// TwinCAT 3 PLC project SEFrey_StringBuilder
// Title: StringBuilder
// Company: S.E.Frey
// Author: Michi
// ProjectVersion: 0.01
// Description: Simple but powerfull stringbuilder, working with any in TC3 available datatype
// ProgramVersion: 3.1.4024.0
// libraries:
//   Tc2_Standard, * (Beckhoff Automation GmbH)
//   Tc2_System, * (Beckhoff Automation GmbH)
//   Tc2_Utilities, * (Beckhoff Automation GmbH)
//   Tc3_Module, * (Beckhoff Automation GmbH)
// project tree:
//   DUTs/ ST_StringBuilderPara.TcDUT
//   GVLs/ GVL_StringBuilder.TcGVL
//   / PlcTask.TcTTO
//   POUs/ MAIN.TcPOU
//   POUs/StringBuilder/ CStringBuilder.TcPOU
//   POUs/StringBuilder/Examples/ CStringBuilderExample.TcPOU
//   POUs/StringBuilder/Functions/ BuildString.TcPOU
//   POUs/StringBuilder/Interfaces/ I_StringBuilder.TcIO
// real-time tasks:
//   TASK PlcTask: cycle T#10ms, priority 20, ADS port 350

CONFIGURATION SEFrey_StringBuilder
    RESOURCE PLC ON TwinCAT3
        TASK PlcTask(INTERVAL := T#10ms, PRIORITY := 20);
        PROGRAM MAIN WITH PlcTask : MAIN;
    END_RESOURCE
END_CONFIGURATION

// ---- DUTs/ST_StringBuilderPara.TcDUT
{attribute 'enable_dynamic_creation'}
TYPE ST_StringBuilderPara :
STRUCT
	MaxBufferSize : UDINT; //defines max possible string length
END_STRUCT
END_TYPE

// ---- GVLs/GVL_StringBuilder.TcGVL
{attribute 'qualified_only'}
VAR_GLOBAL
	pStringBuilder : POINTER TO CStringBuilder;
	pPara : POINTER TO ST_StringBuilderPara;
END_VAR

// ---- POUs/StringBuilder/Interfaces/I_StringBuilder.TcIO
INTERFACE I_StringBuilder

METHOD Append : I_StringBuilder
VAR_INPUT
	Value : T_MaxString;
END_VAR
END_METHOD

METHOD AppendAny : I_StringBuilder
VAR_INPUT
	Value : ANY;
END_VAR
END_METHOD

PROPERTY BufferAddress : POINTER TO BYTE
GET
END_GET
END_PROPERTY

METHOD Clear : I_StringBuilder
VAR_INPUT
END_VAR
END_METHOD

END_INTERFACE

// ---- POUs/MAIN.TcPOU
PROGRAM MAIN
VAR
	StringBuilderExample : CStringBuilderExample;
END_VAR

StringBuilderExample.ClassAndInitialization();
StringBuilderExample.SimpleUse();

END_PROGRAM

// ---- POUs/StringBuilder/Examples/CStringBuilderExample.TcPOU
FUNCTION_BLOCK CStringBuilderExample
VAR_INPUT
END_VAR
VAR_OUTPUT
END_VAR
VAR
	//run tests
	startClassAndInitializationTest, startSimpleUseTest : BOOL;

	
	simpleUseOutput1, simpleUseOutput2 : STRING(200);

	
	StringBuilder : CStringBuilder; //500 characters + 0 terminator (/0)
	Value : STRING(255) := 'Dieser Text ist genau 250 Zeichen lang und wird verwendet, um zu zeigen, wie TwinCAT 3 Strings handhabt. Es handelt sich um einen langen Satz, der viele verschiedene Themen behandelt, wie z.B. Programmierung, Automatisierungstechnik, SPS-Programmieru';
	currentString:  STRING(3000);
	pResult : POINTER TO BYTE;
	Stage, SimpleUseStage : INT;
	
	stStringBuilderPara : ST_StringBuilderPara := (MaxBufferSize:=3000);
	
 	boolExample : BOOL := TRUE;
    byteExample : BYTE := 16#FF;
    wordExample : WORD := 16#FFFF;
    dwordExample : DWORD := 16#FFFFFFFF;
    lwordExample : LWORD := 16#FFFFFFFFFFFFFFFF;
    sintExample : SINT := -128;
    intExample : INT := -32768;
    dintExample : DINT := -2147483648;
    lintExample : LINT := -9223372036854775808;
    usintExample : USINT := 255;
    uintExample : UINT := 65535;
    udintExample : UDINT := 4294967295;
    ulintExample : ULINT := 18446744073709551615;
    realExample : REAL := 1.0;
    lrealExample : LREAL := 1.0;
    timeExample : TIME := T#5s;
    dateExample : DATE := D#2023-01-01;
    todExample : TOD := TOD#12:00:00;
    dtExample : DT := DT#2023-01-01-12:00:00;
    stringExample : STRING := 'I am a string';
END_VAR

METHOD ClassAndInitialization : BOOL
VAR_INPUT
END_VAR
CASE Stage OF
	
	0:
		IF startClassAndInitializationTest THEN
			startClassAndInitializationTest := FALSE;
			StringBUilder.Init(pPara:=ADR(THIS^.stStringBuilderPara));
			Stage := 1;
		END_IF
		
	1:
		StringBuilder
            .Append(Value:='This is a bool: ')
            .AppendAny(Value:=boolExample)
            .Append(Value:=', This is a byte: ')
            .AppendAny(Value:=byteExample)
            .Append(Value:=', This is a word: ')
            .AppendAny(Value:=wordExample)
            .Append(Value:=', This is a dword: ')
            .AppendAny(Value:=dwordExample)
            .Append(Value:=', This is a lword: ')
            .AppendAny(Value:=lwordExample)
            .Append(Value:=', This is a sint: ')
            .AppendAny(Value:=sintExample)
            .Append(Value:=', This is an int: ')
            .AppendAny(Value:=intExample);
			
			//separation done, compiling + logging in needs pretty long for chains longer than 14
			StringBuilder
			.Append(Value:=', This is a dint: ')
            .AppendAny(Value:=dintExample)
            .Append(Value:=', This is a lint: ')
            .AppendAny(Value:=lintExample)
            .Append(Value:=', This is a usint: ')
            .AppendAny(Value:=usintExample)
            .Append(Value:=', This is a uint: ')
            .AppendAny(Value:=uintExample)
            .Append(Value:=', This is a udint: ')
            .AppendAny(Value:=udintExample)
            .Append(Value:=', This is a ulint: ')
            .AppendAny(Value:=ulintExample)
            .Append(Value:=', This is a real: ')
            .AppendAny(Value:=realExample);
			
			StringBuilder
            .Append(Value:=', This is an lreal: ')
            .AppendAny(Value:=lrealExample)
            .Append(Value:=', This is a time: ')
            .AppendAny(Value:=timeExample)
            .Append(Value:=', This is a date: ')
            .AppendAny(Value:=dateExample)
            .Append(Value:=', This is a tod: ')
            .AppendAny(Value:=todExample)
            .Append(Value:=', This is a dt: ')
            .AppendAny(Value:=dtExample)
            .Append(Value:=', This is a string: ')
            .AppendAny(Value:=stringExample);
		// show string data
		StringBuilder.Copy(pDest:=ADR(currentString), n:=SIZEOF(currentString));
		Stage := 2;
		
		2:
			StringBuilder.Clear();
			Stage := 0;
		
		
END_CASE
END_METHOD

METHOD SimpleUse : BOOL
VAR_INPUT
END_VAR
// build string, copy to destination

CASE SimpleUseStage OF


	0:
		IF THIS^.startSimpleUseTest THEN
			startSimpleUseTest := FALSE;
			//build string, copy to given destination
			BuildString(nSizeDest:=SIZEOF(simpleUseOutput1))
			.AppendAny(boolExample)
			.AppendAny(dintExample)
			.Copy(pDest:=ADR(simpleUseOutput1), n:=SIZEOF(simpleUseOutput1));
			SimpleUseStage := 1;
		END_IF
		
	1: //clear buffer, fill + copy to next string
		BuildString(nSizeDest:=SIZEOF(simpleUseOutput2))
		.Clear()
		.AppendAny(dwordExample)
		.AppendAny(dtExample)
		.AppendAny(stringExample)
		.Copy(pDest:=ADR(simpleUseOutput2), n:=SIZEOF(simpleUseOutput2));
		SimpleUseStage := 0;
	
	
	
	
END_CASE
END_METHOD

END_FUNCTION_BLOCK

// ---- POUs/StringBuilder/CStringBuilder.TcPOU
{attribute 'no_assign'}
{attribute 'enable_dynamic_creation'}
{attribute 'no_explicit_call' := 'do not call this POU directly'}
{attribute 'reflection'} 
FUNCTION_BLOCK CStringBuilder IMPLEMENTS I_StringBuilder
VAR_INPUT
END_VAR
VAR_OUTPUT
END_VAR
VAR
	pBuffer : POINTER TO BYTE;
	_maxBufferSize : UDINT; //defines max possible string length
	_currentUsedBufferSize : UDINT;
	
	{attribute 'instance-path'} 
    {attribute 'noinit'} 
    sPath : STRING; 
END_VAR

METHOD AnyToString : STRING
VAR_INPUT
	Value : ANY;
END_VAR
VAR
	pBool			: POINTER TO BOOL;
    pByte			: POINTER TO BYTE;
    pWord			: POINTER TO WORD;
    pDWord			: POINTER TO DWORD;
    pLWord			: POINTER TO LWORD;
    pSint			: POINTER TO SINT;
    pInt			: POINTER TO INT;
    pDint			: POINTER TO DINT;
    pLint			: POINTER TO LINT;
    pUSint			: POINTER TO USINT;
    pUInt			: POINTER TO UINT;
    pUDint			: POINTER TO UDINT;
    pULint			: POINTER TO ULINT;
    pReal			: POINTER TO REAL;
    pLReal			: POINTER TO LREAL;
    pString			: POINTER TO T_MaxString;
    pWString		: POINTER TO WSTRING;
    pTime			: POINTER TO TIME;
    pDate			: POINTER TO DATE;
    pDateAndTime	: POINTER TO DATE_AND_TIME;
    pTimeOfDay		: POINTER TO TIME_OF_DAY;
    pPointer		: PVOID;
	pLTime 			: POINTER TO LTIME;
END_VAR
IF Value.pValue = 0 THEN RETURN; END_IF;

CASE Value.TypeClass OF 
	__SYSTEM.TYPE_CLASS.TYPE_BOOL:
		pBool := Value.pValue;
		AnyToString := TO_STRING(pBool^);
		
    __SYSTEM.TYPE_CLASS.TYPE_BYTE:
		pByte := Value.pValue;
		AnyToString := TO_STRING(pByte^);
		
    __SYSTEM.TYPE_CLASS.TYPE_WORD:
		pWord := Value.pValue;
		AnyToString := TO_STRING(pWord^);
		
    __SYSTEM.TYPE_CLASS.TYPE_DWORD:
		pDWord := Value.pValue;
		AnyToString := TO_STRING(pDWord^);
		
    __SYSTEM.TYPE_CLASS.TYPE_LWORD:
		pLWord := Value.pValue;
		AnyToString := TO_STRING(pLWord^);
		
    __SYSTEM.TYPE_CLASS.TYPE_SINT:
		pSint := Value.pValue;
		AnyToString := TO_STRING(pSint^);
		
    __SYSTEM.TYPE_CLASS.TYPE_INT:
		pInt := Value.pValue;
		AnyToString := TO_STRING(pInt^);
		
    __SYSTEM.TYPE_CLASS.TYPE_DINT:
		pDint := Value.pValue;
		AnyToString := TO_STRING(pDint^);
		
    __SYSTEM.TYPE_CLASS.TYPE_LINT:
		pLint := Value.pValue;
		AnyToString := TO_STRING(pLint^);
		
    __SYSTEM.TYPE_CLASS.TYPE_USINT:
		pUSint := Value.pValue;
		AnyToString := TO_STRING(pUSint^);
		
    __SYSTEM.TYPE_CLASS.TYPE_UINT:
		pUInt := Value.pValue;
		AnyToString := TO_STRING(pUInt^);
		
    __SYSTEM.TYPE_CLASS.TYPE_UDINT:
		pUDint := Value.pValue;
		AnyToString := TO_STRING(pUDint^);
		
    __SYSTEM.TYPE_CLASS.TYPE_ULINT:
		pULint := Value.pValue;
		AnyToString := TO_STRING(pULint^);
		
   __SYSTEM.TYPE_CLASS.TYPE_REAL:
		pReal := Value.pValue;
		AnyToString := TO_STRING(pReal^);
		
    __SYSTEM.TYPE_CLASS.TYPE_LREAL:
		pLReal := Value.pValue;
		AnyToString := TO_STRING(pLReal^);
		
    __SYSTEM.TYPE_CLASS.TYPE_STRING:
		pString := Value.pValue;
		AnyToString := TO_STRING(pString^);
		
   __SYSTEM.TYPE_CLASS.TYPE_WSTRING:
		pWString := Value.pValue;
		AnyToString := TO_STRING(pWString^);
		
    __SYSTEM.TYPE_CLASS.TYPE_TIME:
		pTime := Value.pValue;
		AnyToString := TO_STRING(pTime^);
		
    __SYSTEM.TYPE_CLASS.TYPE_DATE:
		pDate := Value.pValue;
		AnyToString := TO_STRING(pDate^);
		
    __SYSTEM.TYPE_CLASS.TYPE_DATEANDTIME:
		pDateAndTime := Value.pValue;
		AnyToString := TO_STRING(pDateAndTime^);
		
    __SYSTEM.TYPE_CLASS.TYPE_TIMEOFDAY:
		pTimeOfDay := Value.pValue;
		AnyToString := TO_STRING(pTimeOfDay^);
	
	__SYSTEM.TYPE_CLASS.TYPE_POINTER:
		AnyToString := TO_STRING(Value.pValue);
		
	__SYSTEM.TYPE_CLASS.TYPE_LTIME:
		pLTime := Value.pValue;
		AnyToString := TO_STRING(pLTime^);
ELSE
	RETURN; 
END_CASE
END_METHOD

METHOD Append : I_StringBuilder
VAR_INPUT
	Value : T_MaxString;
END_VAR
Append := THIS^.AppendAny(Value);
END_METHOD

// Appends the given value to the end of the string builder's contents.
METHOD AppendAny : I_StringBuilder
VAR_INPUT
	Value : ANY;
END_VAR
VAR
	stringLength : UDINT;
	convertedAny : STRING; 
	pValue : POINTER TO BYTE;
END_VAR
AppendAny := THIS^;

IF THIS^.pBuffer = 0 THEN
	ADSLOGSTR(msgCtrlMask:= ADSLOG_MSGTYPE_ERROR, msgFmtStr:='Dynamic buffer null pointer, usage of StringBuilder not possible', '');
	RETURN;
END_IF

CASE Value.TypeClass OF
	__SYSTEM.TYPE_CLASS.TYPE_STRING: 
		pValue := Value.pValue;
		
	__SYSTEM.TYPE_CLASS.TYPE_BOOL,
	__SYSTEM.TYPE_CLASS.TYPE_BYTE,
	__SYSTEM.TYPE_CLASS.TYPE_WORD,
	__SYSTEM.TYPE_CLASS.TYPE_DWORD,
	__SYSTEM.TYPE_CLASS.TYPE_LWORD,
	__SYSTEM.TYPE_CLASS.TYPE_SINT,
	__SYSTEM.TYPE_CLASS.TYPE_INT,
	__SYSTEM.TYPE_CLASS.TYPE_DINT,
	__SYSTEM.TYPE_CLASS.TYPE_LINT,
	__SYSTEM.TYPE_CLASS.TYPE_USINT,
	__SYSTEM.TYPE_CLASS.TYPE_UINT,
	__SYSTEM.TYPE_CLASS.TYPE_UDINT,
	__SYSTEM.TYPE_CLASS.TYPE_ULINT,
	__SYSTEM.TYPE_CLASS.TYPE_REAL,
	__SYSTEM.TYPE_CLASS.TYPE_LREAL,
	__SYSTEM.TYPE_CLASS.TYPE_TIME,
	__SYSTEM.TYPE_CLASS.TYPE_LTIME,
	__SYSTEM.TYPE_CLASS.TYPE_DATE,
	__SYSTEM.TYPE_CLASS.TYPE_DATEANDTIME,
	__SYSTEM.TYPE_CLASS.TYPE_TIMEOFDAY,
	__SYSTEM.TYPE_CLASS.TYPE_POINTER:
		convertedAny := AnyToString(Value);
		pValue := ADR(convertedAny);
ELSE
	RETURN;
END_CASE

stringLength := GetUsedStringLength(pByte:=pValue);

//check available size, existing size
IF stringLength = 0 THEN
	RETURN;
END_IF
//only copy if we do not exceed possible limit
IF THIS^._currentUsedBufferSize + stringLength >= THIS^._maxBufferSize THEN
	RETURN;
END_IF
MEMCPY(destAddr:=(THIS^.pBuffer + THIS^._currentUsedBufferSize), srcAddr:=pValue, n:=stringLength);

THIS^._currentUsedBufferSize := THIS^._currentUsedBufferSize + stringLength;
END_METHOD

PROPERTY BufferAddress : POINTER TO BYTE
GET
BufferAddress := THIS^.pBuffer;
END_GET
END_PROPERTY

METHOD Clear : I_StringBuilder
VAR_INPUT
END_VAR
Clear := THIS^;
IF THIS^.pBuffer = 0 THEN
	RETURN;
END_IF

MEMSET(destAddr:=THIS^.pBuffer, fillByte:=0, n:=THIS^.MaxBufferSize);
_currentUsedBufferSize := 0;
END_METHOD

METHOD Copy : BOOL
VAR_INPUT
	pDest : POINTER TO BYTE;
	n : UDINT; // Size of destination
END_VAR
MEMCPY(destAddr:=pDest, srcAddr:=THIS^.BufferAddress, n:=n);
Copy := TRUE;
END_METHOD

PROPERTY CurrentBufferSize : UDINT
GET
CurrentBufferSize := THIS^._currentUsedBufferSize;
END_GET
END_PROPERTY

METHOD GetUsedStringLength : UDINT
VAR_INPUT
	pByte : POINTER TO BYTE;
END_VAR
VAR
    i : UDINT := 0;
END_VAR
//every string in twincat is 0 terminated
IF pByte = 0 THEN
	RETURN;
END_IF

WHILE (pByte^ <> 0) DO
    pByte := pByte + 1; // Pointer auf das nächste Byte verschieben
    i := i + 1;
END_WHILE;

GetUsedStringLength := i;
END_METHOD

METHOD Init : I_StringBuilder
VAR_INPUT
	pPara : POINTER TO ST_StringBuilderPara;
END_VAR
// TODO: add logging for failed allocation
IF ParaErrors(pPara:=pPara) THEN
	RETURN;
END_IF

IF THIS^.pBuffer <> 0 THEN
	__DELETE(THIS^.pBuffer);
END_IF

THIS^.pBuffer := __NEW(BYTE, pPara^.MaxBufferSize);
THIS^._maxBufferSize := pPara^.MaxBufferSize;
END_METHOD

PROPERTY MaxBufferSize : UDINT
GET
MaxBufferSize := THIS^._maxBufferSize;
END_GET
END_PROPERTY

{attribute 'reflection'} 
METHOD PRIVATE ParaErrors : BOOL
VAR_INPUT
	pPara : POINTER TO ST_StringBuilderPara;
END_VAR
VAR
	s1 : STRING(35) := 'Invalid parametrization pointer at ';
	s2: T_MaxString;
END_VAR
IF pPara = 0 THEN
	CONCAT2(pSrcString1:=ADR(s1), pSrcString2:=ADR(THIS^.sPath), pDstString:=ADR(s2), nDstSize:=SIZEOF(s2));
	ADSLOGSTR(msgCtrlMask:= ADSLOG_MSGTYPE_ERROR, msgFmtStr:=s2, '');
	ParaErrors := TRUE;
	RETURN;
END_IF
IF pPara^.MaxBufferSize = 0 THEN
	s1 := 'BufferSize 0 given, Stringbuilder init failed at ';
	CONCAT2(pSrcString1:=ADR(s1), pSrcString2:=ADR(THIS^.sPath), pDstString:=ADR(s2), nDstSize:=SIZEOF(s2));
	ADSLOGSTR(msgCtrlMask:= ADSLOG_MSGTYPE_ERROR, msgFmtStr:=s2, '');
	ParaErrors := TRUE;
	RETURN;
END_IF
END_METHOD

METHOD Reset : I_StringBuilder
VAR_INPUT
	pPara : POINTER TO ST_StringBuilderPara;
END_VAR
Reset := THIS^;
Clear();

IF ParaErrors(pPara:=pPara) THEN
	RETURN;
END_IF

Init(pPara:=pPara);
END_METHOD

END_FUNCTION_BLOCK

// ---- POUs/StringBuilder/Functions/BuildString.TcPOU
//simple function use without insantiation
FUNCTION BuildString : I_StringBuilder
VAR_INPUT
	nSizeDest : UDINT;
END_VAR
VAR
END_VAR

IF nSizeDest = 0 THEN
	RETURN;
END_IF

//Create if nonExistend
IF GVL_StringBuilder.pStringBuilder = 0 THEN
	GVL_StringBuilder.pStringBuilder := __NEW(CStringbuilder);
END_IF

// TODO: zero interface return
IF GVL_StringBuilder.pStringBuilder = 0 THEN
	ADSLOGSTR(msgCtrlMask:= ADSLOG_MSGTYPE_ERROR, msgFmtStr:='StringBuilder creation for GVL_StringBuilder failed', '');
	RETURN;
END_IF

IF GVL_StringBuilder.pPara = 0 THEN
	GVL_StringBuilder.pPara := __NEW(ST_StringBuilderPara);
END_IF

// TODO: zero interface return
IF GVL_StringBuilder.pPara = 0 THEN
	ADSLOGSTR(msgCtrlMask:= ADSLOG_MSGTYPE_ERROR, msgFmtStr:='ST_Para for GVL_StringBuilder failed', '');
	RETURN;
END_IF

GVL_StringBuilder.pPara^.MaxBufferSize := nSizeDest;

// adapt needed bufferSize
IF nSizeDest > GVL_StringBuilder.pStringBuilder^.MaxBufferSize THEN
	GVL_StringBuilder.pStringBuilder^.Reset(pPara:=GVL_StringBuilder.pPara);
END_IF


BuildString := GVL_StringBuilder.pStringBuilder^;

END_FUNCTION
